FUNCTION_BLOCK FT_PIDWL (* PI Controller with Anti-Windup *)
  (* Standard: 61499-1; Description: version 1.3	13. nov. 2009 programmer 	hugo tested by		tobias FT_PIDWL is a PID controller with dynamic wind_up reset. The PID controller works according to the fomula Y = KP *(IN + KI * INTEG(e) + DERIV(e) ). a rst will reset the integrator to 0 lim_h and Lim_l set the possible output range of the internal integrator. the output flags lim will signal that the output limits are active. *)
  (* Version 1.0, 2025-12-19, franz *)
  PACKAGE OSCAT::Basic::POUs::Engineering::Control;
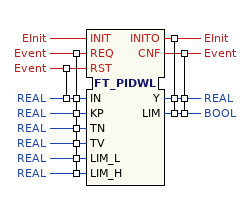
  EVENT_INPUT
    INIT : EInit; (* Init Request *)
    REQ WITH IN, KP, TN, TV, LIM_L, LIM_H; (* Normal Execution Request *)
    RST WITH IN; (* Reset Integrator *)
  END_EVENT
  EVENT_OUTPUT
    INITO : EInit WITH Y, LIM; (* Init Confirmation *)
    CNF WITH Y, LIM; (* Execution Confirmation *)
  END_EVENT
  VAR_INPUT
    IN : REAL; (* Process Variable Input *)
    KP : REAL := 1.0; (* Proportional Gain *)
    TN : REAL := 1.0; (* Integral Time *)
    TV : REAL := 1.0; (* Derivative Time *)
    LIM_L : REAL := -1.0E38; (* Output Limit Low *)
    LIM_H : REAL := 1.0E38; (* Output Limit High *)
  END_VAR
  VAR_OUTPUT
    Y : REAL; (* PID Output *)
    LIM : BOOL; (* Limit reached flag *)
  END_VAR
  FBS
    piwl : OSCAT::Basic::POUs::Engineering::Control::FT_PIWL; (* Internal PI Controller *)
    diff : OSCAT::Basic::POUs::Engineering::Control::FT_DERIV; (* Internal Differentiator *)
  END_FBS
  EC_STATES
    INIT : INIT -> INITO;
    REQ : REQ -> CNF;
    RST : RST -> CNF;
  END_STATES
  ALGORITHM INIT IN ST:
(* Init internal instances if necessary, typically empty or reset logic *)
piwl.INIT();
diff.INIT(); (* Initialize diff input *)
Y := 0.0;
LIM := FALSE;
  END_ALGORITHM
  ALGORITHM RST IN ST:
piwl.RST();
  END_ALGORITHM
  ALGORITHM REQ IN ST:
ALGORITHM REQ
(* run PIWL controller first *)
(* we need to check if TN = 0 and do alternative calls *)
IF TN = 0.0 THEN
	piwl.REQ(in := IN * KP, KP := 1.0, KI := 0.0, LIM_L := LIM_L, LIM_H := LIM_H);
ELSE
	piwl.REQ(in := IN * KP, KP := 1.0, KI := 1.0 / TN, LIM_L := LIM_L, LIM_H := LIM_H);
END_IF;

(* run differentiator and add_to_output *)
diff.REQ(IN := IN, K := KP * TV);
Y := piwl.Y + diff.out;

(* limit the output *)
IF Y < LIM_L THEN
	LIM := TRUE;
	Y := LIM_L;
ELSIF Y > LIM_H THEN
	LIM := TRUE;
	Y := LIM_H;
ELSE
	LIM := FALSE;
END_IF;
END_ALGORITHM

(* revision history hm 13. jun. 2008 	rev 1.0 original version
 * *
 * hm	25. jan 2008	rev 1.1 multiply differential part with KP
 * *
 * hm	11. mar. 2009	rev 1.2 real constants updated to new systax using dot
 * *
 * hm	13. nov. 2009	rev 1.3 fixed code for negative KP *)
  END_ALGORITHM
END_FUNCTION_BLOCK
